(* IEC 61131-3 sources: IRIS-Project/LASAL CONTROL SOFTWARE/LasalProject_2025_09_12/Class/QuitError, 1 file *)

(* ---- QuitError.st ---- *)
(*!
<Class
	Name               = "QuitError"
	Revision           = "0.0"
	RealtimeTask       = "false"
	CyclicTask         = "true"
	DefCyclictime      = "100 ms"
	BackgroundTask     = "false"
	Sigmatek           = "false"
	OSInterface        = "false"
	HighPriority       = "false"
	Automatic          = "false"
	UpdateMode         = "Prescan"
	SharedCommandTable = "true"
	Objectsize         = "(284,120)">
	<Channels>
		<Server Name="ClassSvr" Visualized="false" Initialize="false" WriteProtected="true" Retentive="false"/>
		<Client Name="M1" Required="true" Internal="false"/>
	</Channels>
</Class>
*)
QuitError : CLASS
  //Servers:
	ClassSvr 	: SvrChCmd_DINT;
  //Clients:
	M1 	: CltChCmd__LMCAxisBase;
  //Variables:
		A 	: DINT;
  //Functions:

	FUNCTION VIRTUAL GLOBAL Init;

	FUNCTION VIRTUAL GLOBAL CyWork
		VAR_INPUT
			EAX 	: UDINT;
		END_VAR
		VAR_OUTPUT
			state (EAX) 	: UDINT;
		END_VAR;

	FUNCTION GLOBAL ResetAll
		VAR_INPUT
			Input 	: DINT;
		END_VAR;
  //Tables:
	FUNCTION @STD
		VAR_OUTPUT
			ret_code	: CONFSTATES;
		END_VAR;
	FUNCTION GLOBAL TAB @CT_;
END_CLASS;

#pragma usingLtd _LMCAxisBase

FUNCTION VIRTUAL GLOBAL QuitError::CyWork
	VAR_INPUT
		EAX 	: UDINT;
	END_VAR
	VAR_OUTPUT
		state (EAX) 	: UDINT;
	END_VAR

  if A=1 then
M1.QuitError();
  end_if;

	state := READY;

END_FUNCTION

FUNCTION GLOBAL QuitError::ResetAll
	VAR_INPUT
		Input 	: DINT;
	END_VAR
A:=Input;
END_FUNCTION

FUNCTION VIRTUAL GLOBAL QuitError::Init
A:=0;
END_FUNCTION
